Fanuc KAREL source: ks00040.KL

-- PROVISIONAL review KL for V770-1; original PC SHA256 47b8b368d995e283385770092253cdfeffd99626a467b9d59ca32cd929f8968e
-- Incomplete behavior may be omitted. Consult companion uncertainty JSON. Do not deploy.
PROGRAM KS00040
%NOLOCKGROUP
BEGIN
  -- UNRESOLVED_PC offsets 5-13; opcodes 3F,75
  -- UNRESOLVED_PC offsets 18-27; opcodes 3F,75
  -- UNRESOLVED_PC offsets 32-45; opcodes 22,1D,23
  -- UNRESOLVED_PC offsets 50-54; opcodes 7F
END KS00040
